// TIA Portal V21 export
FUNCTION "AlarmsFc" : Void   // FC181, LAD
{ S7_Optimized_Access := 'TRUE' }
// stored: AutoNumber false, SetENOAutomatically false
   VAR_TEMP   // added for the SCL form of the ladder/FBD networks
      _w1 : Bool;
      _w2 : Bool;
      _w3 : Bool;
      _w4 : Bool;
      _w5 : Bool;
      _w6 : Bool;
      _w7 : Bool;
      _w8 : Bool;
      _w9 : Bool;
      _w10 : Bool;
      _w11 : Bool;
      _w12 : Bool;
      _w13 : Bool;
      _w14 : Bool;
      _w15 : Bool;
      _w16 : Bool;
      _w17 : Bool;
      _w18 : Bool;
      _w19 : Bool;
      _w20 : Bool;
      _w21 : Bool;
      _w22 : Bool;
      _w23 : Bool;
      _w24 : Bool;
      _w25 : Bool;
      _w26 : Bool;
      _w27 : Bool;
      _w28 : Bool;
      _w29 : Bool;
      _w30 : Bool;
      _w31 : Bool;
      _w32 : Bool;
      _w33 : Bool;
      _w34 : Bool;
      _w35 : Bool;
      _w36 : Bool;
      _w37 : Bool;
      _w38 : Bool;
      _w39 : Bool;
      _w40 : Bool;
      _w41 : Bool;
      _w42 : Bool;
      _w43 : Bool;
      _w44 : Bool;
      _w45 : Bool;
      _w46 : Bool;
   END_VAR
BEGIN

REGION Network 1: "SafetyAlarms".ControlKeyOff
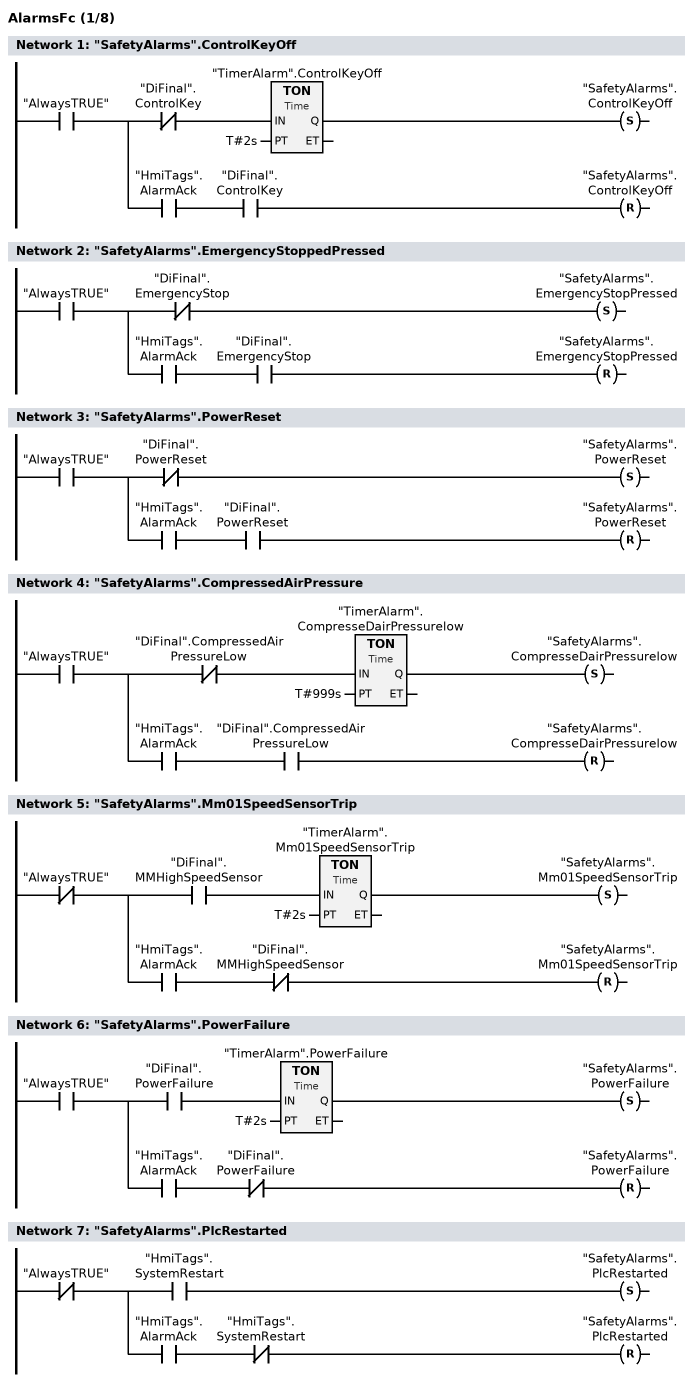
   RUNG wire#powerrail
      Contact( "AlwaysTRUE" )
      wire#w1
      I_Contact( "DiFinal".ControlKey )
      { S7_Templates := "time_type := Time" } "TimerAlarm".ControlKeyOff.TON(pt := T#2s, et =>)
      S_Coil( "SafetyAlarms".ControlKeyOff )
   END_RUNG
   RUNG wire#w1
      Contact( "HmiTags".AlarmAck )
      Contact( "DiFinal".ControlKey )
      R_Coil( "SafetyAlarms".ControlKeyOff )
   END_RUNG
   // the same network as SCL:
   "TimerAlarm".ControlKeyOff.TON(IN := "AlwaysTRUE" AND NOT "DiFinal".ControlKey, PT := T#2s);
   IF "TimerAlarm".ControlKeyOff.Q THEN "SafetyAlarms".ControlKeyOff := TRUE; END_IF;
   IF "AlwaysTRUE" AND "HmiTags".AlarmAck AND "DiFinal".ControlKey THEN
       "SafetyAlarms".ControlKeyOff := FALSE;
   END_IF;
END_REGION

REGION Network 2: "SafetyAlarms".EmergencyStoppedPressed
   RUNG wire#powerrail
      Contact( "AlwaysTRUE" )
      wire#w1
      I_Contact( "DiFinal".EmergencyStop )
      S_Coil( "SafetyAlarms".EmergencyStopPressed )
   END_RUNG
   RUNG wire#w1
      Contact( "HmiTags".AlarmAck )
      Contact( "DiFinal".EmergencyStop )
      R_Coil( "SafetyAlarms".EmergencyStopPressed )
   END_RUNG
   // the same network as SCL:
   IF "AlwaysTRUE" AND NOT "DiFinal".EmergencyStop THEN "SafetyAlarms".EmergencyStopPressed := TRUE; END_IF;
   IF "AlwaysTRUE" AND "HmiTags".AlarmAck AND "DiFinal".EmergencyStop THEN
       "SafetyAlarms".EmergencyStopPressed := FALSE;
   END_IF;
END_REGION

REGION Network 3: "SafetyAlarms".PowerReset
   RUNG wire#powerrail
      Contact( "AlwaysTRUE" )
      wire#w1
      I_Contact( "DiFinal".PowerReset )
      S_Coil( "SafetyAlarms".PowerReset )
   END_RUNG
   RUNG wire#w1
      Contact( "HmiTags".AlarmAck )
      Contact( "DiFinal".PowerReset )
      R_Coil( "SafetyAlarms".PowerReset )
   END_RUNG
   // the same network as SCL:
   IF "AlwaysTRUE" AND NOT "DiFinal".PowerReset THEN "SafetyAlarms".PowerReset := TRUE; END_IF;
   IF "AlwaysTRUE" AND "HmiTags".AlarmAck AND "DiFinal".PowerReset THEN
       "SafetyAlarms".PowerReset := FALSE;
   END_IF;
END_REGION

REGION Network 4: "SafetyAlarms".CompressedAirPressure
   RUNG wire#powerrail
      Contact( "AlwaysTRUE" )
      wire#w1
      I_Contact( "DiFinal".CompressedAirPressureLow )
      { S7_Templates := "time_type := Time" } "TimerAlarm".CompresseDairPressurelow.TON(pt := T#999s, et =>)
      S_Coil( "SafetyAlarms".CompresseDairPressurelow )
   END_RUNG
   RUNG wire#w1
      Contact( "HmiTags".AlarmAck )
      Contact( "DiFinal".CompressedAirPressureLow )
      R_Coil( "SafetyAlarms".CompresseDairPressurelow )
   END_RUNG
   // the same network as SCL:
   "TimerAlarm".CompresseDairPressurelow.TON(IN := "AlwaysTRUE" AND NOT "DiFinal".CompressedAirPressureLow,
                           PT := T#999s);
   IF "TimerAlarm".CompresseDairPressurelow.Q THEN "SafetyAlarms".CompresseDairPressurelow := TRUE; END_IF;
   IF "AlwaysTRUE" AND "HmiTags".AlarmAck AND "DiFinal".CompressedAirPressureLow THEN
       "SafetyAlarms".CompresseDairPressurelow := FALSE;
   END_IF;
END_REGION

REGION Network 5: "SafetyAlarms".Mm01SpeedSensorTrip
   RUNG wire#powerrail
      I_Contact( "AlwaysTRUE" )
      wire#w1
      Contact( "DiFinal".MMHighSpeedSensor )
      { S7_Templates := "time_type := Time" } "TimerAlarm".Mm01SpeedSensorTrip.TON(pt := T#2s, et =>)
      S_Coil( "SafetyAlarms".Mm01SpeedSensorTrip )
   END_RUNG
   RUNG wire#w1
      Contact( "HmiTags".AlarmAck )
      I_Contact( "DiFinal".MMHighSpeedSensor )
      R_Coil( "SafetyAlarms".Mm01SpeedSensorTrip )
   END_RUNG
   // the same network as SCL:
   "TimerAlarm".Mm01SpeedSensorTrip.TON(IN := NOT "AlwaysTRUE" AND "DiFinal".MMHighSpeedSensor, PT := T#2s);
   IF "TimerAlarm".Mm01SpeedSensorTrip.Q THEN "SafetyAlarms".Mm01SpeedSensorTrip := TRUE; END_IF;
   IF NOT "AlwaysTRUE" AND "HmiTags".AlarmAck AND NOT "DiFinal".MMHighSpeedSensor THEN
       "SafetyAlarms".Mm01SpeedSensorTrip := FALSE;
   END_IF;
END_REGION

REGION Network 6: "SafetyAlarms".PowerFailure
   RUNG wire#powerrail
      Contact( "AlwaysTRUE" )
      wire#w1
      Contact( "DiFinal".PowerFailure )
      { S7_Templates := "time_type := Time" } "TimerAlarm".PowerFailure.TON(pt := T#2s, et =>)
      S_Coil( "SafetyAlarms".PowerFailure )
   END_RUNG
   RUNG wire#w1
      Contact( "HmiTags".AlarmAck )
      I_Contact( "DiFinal".PowerFailure )
      R_Coil( "SafetyAlarms".PowerFailure )
   END_RUNG
   // the same network as SCL:
   "TimerAlarm".PowerFailure.TON(IN := "AlwaysTRUE" AND "DiFinal".PowerFailure, PT := T#2s);
   IF "TimerAlarm".PowerFailure.Q THEN "SafetyAlarms".PowerFailure := TRUE; END_IF;
   IF "AlwaysTRUE" AND "HmiTags".AlarmAck AND NOT "DiFinal".PowerFailure THEN
       "SafetyAlarms".PowerFailure := FALSE;
   END_IF;
END_REGION

REGION Network 7: "SafetyAlarms".PlcRestarted
   RUNG wire#powerrail
      I_Contact( "AlwaysTRUE" )
      wire#w1
      Contact( "HmiTags".SystemRestart )
      S_Coil( "SafetyAlarms".PlcRestarted )
   END_RUNG
   RUNG wire#w1
      Contact( "HmiTags".AlarmAck )
      I_Contact( "HmiTags".SystemRestart )
      R_Coil( "SafetyAlarms".PlcRestarted )
   END_RUNG
   // the same network as SCL:
   IF NOT "AlwaysTRUE" AND "HmiTags".SystemRestart THEN "SafetyAlarms".PlcRestarted := TRUE; END_IF;
   IF NOT "AlwaysTRUE" AND "HmiTags".AlarmAck AND NOT "HmiTags".SystemRestart THEN
       "SafetyAlarms".PlcRestarted := FALSE;
   END_IF;
END_REGION

REGION Network 8: "SafetyAlarms".Mm01OverloadTrip
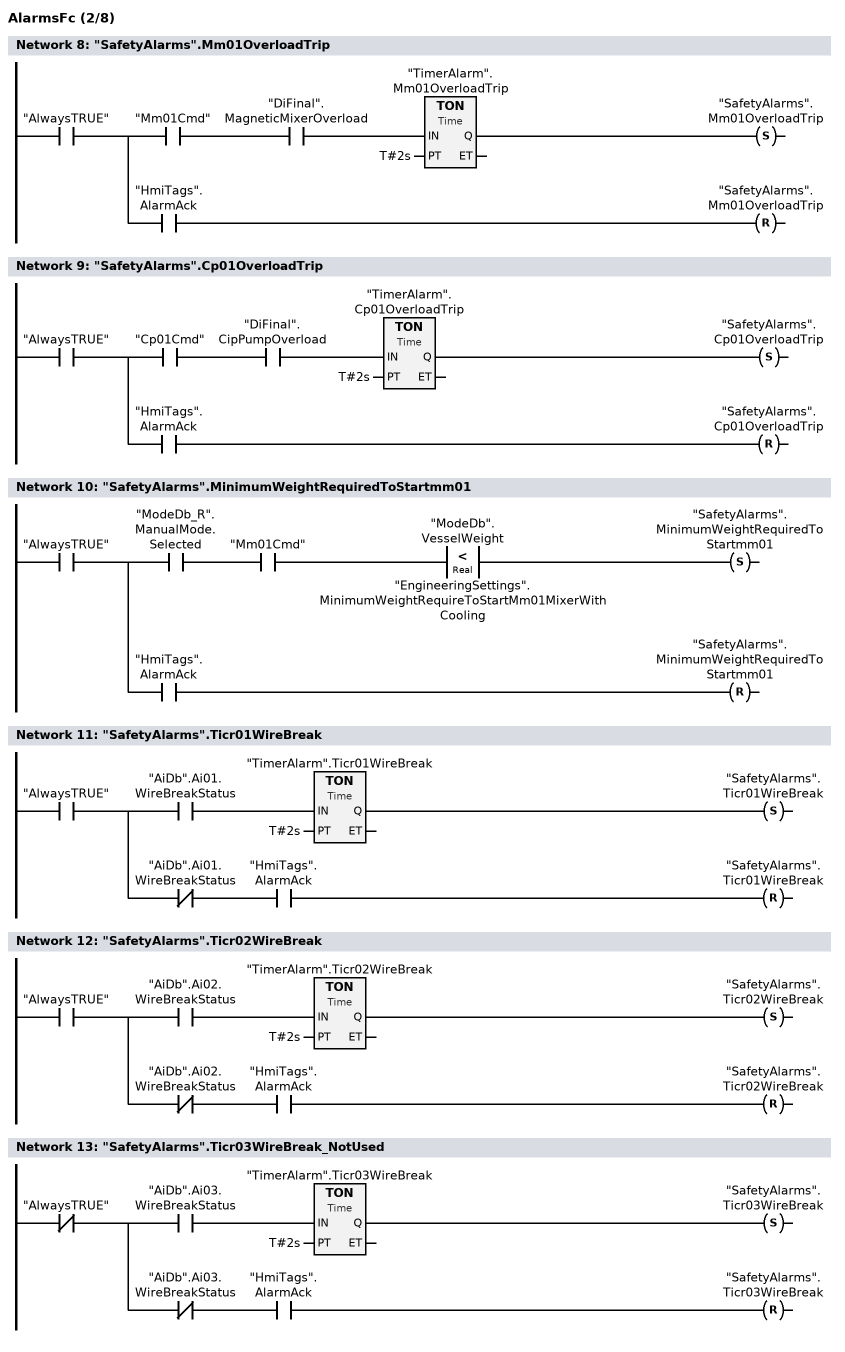
   RUNG wire#powerrail
      Contact( "AlwaysTRUE" )
      wire#w1
      Contact( "Mm01Cmd" )
      Contact( "DiFinal".MagneticMixerOverload )
      { S7_Templates := "time_type := Time" } "TimerAlarm".Mm01OverloadTrip.TON(pt := T#2s, et =>)
      S_Coil( "SafetyAlarms".Mm01OverloadTrip )
   END_RUNG
   RUNG wire#w1
      Contact( "HmiTags".AlarmAck )
      R_Coil( "SafetyAlarms".Mm01OverloadTrip )
   END_RUNG
   // the same network as SCL:
   "TimerAlarm".Mm01OverloadTrip.TON(IN := "AlwaysTRUE" AND "Mm01Cmd" AND "DiFinal".MagneticMixerOverload,
                           PT := T#2s);
   IF "TimerAlarm".Mm01OverloadTrip.Q THEN "SafetyAlarms".Mm01OverloadTrip := TRUE; END_IF;
   IF "AlwaysTRUE" AND "HmiTags".AlarmAck THEN "SafetyAlarms".Mm01OverloadTrip := FALSE; END_IF;
END_REGION

REGION Network 9: "SafetyAlarms".Cp01OverloadTrip
   RUNG wire#powerrail
      Contact( "AlwaysTRUE" )
      wire#w1
      Contact( "Cp01Cmd" )
      Contact( "DiFinal".CipPumpOverload )
      { S7_Templates := "time_type := Time" } "TimerAlarm".Cp01OverloadTrip.TON(pt := T#2s, et =>)
      S_Coil( "SafetyAlarms".Cp01OverloadTrip )
   END_RUNG
   RUNG wire#w1
      Contact( "HmiTags".AlarmAck )
      R_Coil( "SafetyAlarms".Cp01OverloadTrip )
   END_RUNG
   // the same network as SCL:
   "TimerAlarm".Cp01OverloadTrip.TON(IN := "AlwaysTRUE" AND "Cp01Cmd" AND "DiFinal".CipPumpOverload, PT := T#2s);
   IF "TimerAlarm".Cp01OverloadTrip.Q THEN "SafetyAlarms".Cp01OverloadTrip := TRUE; END_IF;
   IF "AlwaysTRUE" AND "HmiTags".AlarmAck THEN "SafetyAlarms".Cp01OverloadTrip := FALSE; END_IF;
END_REGION

REGION Network 10: "SafetyAlarms".MinimumWeightRequiredToStartmm01
   RUNG wire#powerrail
      Contact( "AlwaysTRUE" )
      wire#w1
      Contact( "ModeDb_R".ManualMode.Selected )
      Contact( "Mm01Cmd" )
      { S7_Templates := "SrcType := Real" } LT_Contact(in1 := "ModeDb".VesselWeight, in2 := "EngineeringSettings".MinimumWeightRequireToStartMm01MixerWithCooling)
      S_Coil( "SafetyAlarms".MinimumWeightRequiredToStartmm01 )
   END_RUNG
   RUNG wire#w1
      Contact( "HmiTags".AlarmAck )
      R_Coil( "SafetyAlarms".MinimumWeightRequiredToStartmm01 )
   END_RUNG
   // the same network as SCL:
   IF "AlwaysTRUE" AND "ModeDb_R".ManualMode.Selected AND "Mm01Cmd" AND ("ModeDb".VesselWeight < "EngineeringSettings".MinimumWeightRequireToStartMm01MixerWithCooling) THEN
       "SafetyAlarms".MinimumWeightRequiredToStartmm01 := TRUE;
   END_IF;
   IF "AlwaysTRUE" AND "HmiTags".AlarmAck THEN
       "SafetyAlarms".MinimumWeightRequiredToStartmm01 := FALSE;
   END_IF;
END_REGION

REGION Network 11: "SafetyAlarms".Ticr01WireBreak
   RUNG wire#powerrail
      Contact( "AlwaysTRUE" )
      wire#w1
      Contact( "AiDb".Ai01.WireBreakStatus )
      { S7_Templates := "time_type := Time" } "TimerAlarm".Ticr01WireBreak.TON(pt := T#2s, et =>)
      S_Coil( "SafetyAlarms".Ticr01WireBreak )
   END_RUNG
   RUNG wire#w1
      I_Contact( "AiDb".Ai01.WireBreakStatus )
      Contact( "HmiTags".AlarmAck )
      R_Coil( "SafetyAlarms".Ticr01WireBreak )
   END_RUNG
   // the same network as SCL:
   "TimerAlarm".Ticr01WireBreak.TON(IN := "AlwaysTRUE" AND "AiDb".Ai01.WireBreakStatus, PT := T#2s);
   IF "TimerAlarm".Ticr01WireBreak.Q THEN "SafetyAlarms".Ticr01WireBreak := TRUE; END_IF;
   IF "AlwaysTRUE" AND NOT "AiDb".Ai01.WireBreakStatus AND "HmiTags".AlarmAck THEN
       "SafetyAlarms".Ticr01WireBreak := FALSE;
   END_IF;
END_REGION

REGION Network 12: "SafetyAlarms".Ticr02WireBreak
   RUNG wire#powerrail
      Contact( "AlwaysTRUE" )
      wire#w1
      Contact( "AiDb".Ai02.WireBreakStatus )
      { S7_Templates := "time_type := Time" } "TimerAlarm".Ticr02WireBreak.TON(pt := T#2s, et =>)
      S_Coil( "SafetyAlarms".Ticr02WireBreak )
   END_RUNG
   RUNG wire#w1
      I_Contact( "AiDb".Ai02.WireBreakStatus )
      Contact( "HmiTags".AlarmAck )
      R_Coil( "SafetyAlarms".Ticr02WireBreak )
   END_RUNG
   // the same network as SCL:
   "TimerAlarm".Ticr02WireBreak.TON(IN := "AlwaysTRUE" AND "AiDb".Ai02.WireBreakStatus, PT := T#2s);
   IF "TimerAlarm".Ticr02WireBreak.Q THEN "SafetyAlarms".Ticr02WireBreak := TRUE; END_IF;
   IF "AlwaysTRUE" AND NOT "AiDb".Ai02.WireBreakStatus AND "HmiTags".AlarmAck THEN
       "SafetyAlarms".Ticr02WireBreak := FALSE;
   END_IF;
END_REGION

REGION Network 13: "SafetyAlarms".Ticr03WireBreak_NotUsed
   RUNG wire#powerrail
      I_Contact( "AlwaysTRUE" )
      wire#w1
      Contact( "AiDb".Ai03.WireBreakStatus )
      { S7_Templates := "time_type := Time" } "TimerAlarm".Ticr03WireBreak.TON(pt := T#2s, et =>)
      S_Coil( "SafetyAlarms".Ticr03WireBreak )
   END_RUNG
   RUNG wire#w1
      I_Contact( "AiDb".Ai03.WireBreakStatus )
      Contact( "HmiTags".AlarmAck )
      R_Coil( "SafetyAlarms".Ticr03WireBreak )
   END_RUNG
   // the same network as SCL:
   "TimerAlarm".Ticr03WireBreak.TON(IN := NOT "AlwaysTRUE" AND "AiDb".Ai03.WireBreakStatus, PT := T#2s);
   IF "TimerAlarm".Ticr03WireBreak.Q THEN "SafetyAlarms".Ticr03WireBreak := TRUE; END_IF;
   IF NOT "AlwaysTRUE" AND NOT "AiDb".Ai03.WireBreakStatus AND "HmiTags".AlarmAck THEN
       "SafetyAlarms".Ticr03WireBreak := FALSE;
   END_IF;
END_REGION

REGION Network 14: "SafetyAlarms".Ticr04WireBreak_NotUsed
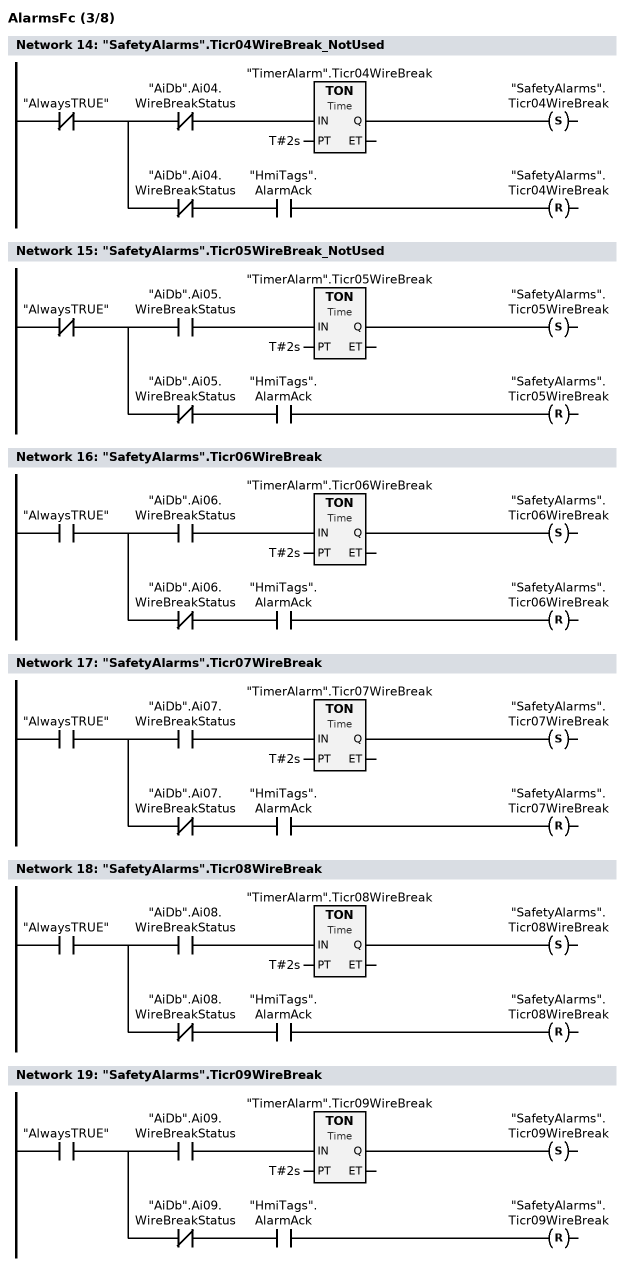
   RUNG wire#powerrail
      I_Contact( "AlwaysTRUE" )
      wire#w1
      I_Contact( "AiDb".Ai04.WireBreakStatus )
      { S7_Templates := "time_type := Time" } "TimerAlarm".Ticr04WireBreak.TON(pt := T#2s, et =>)
      S_Coil( "SafetyAlarms".Ticr04WireBreak )
   END_RUNG
   RUNG wire#w1
      I_Contact( "AiDb".Ai04.WireBreakStatus )
      Contact( "HmiTags".AlarmAck )
      R_Coil( "SafetyAlarms".Ticr04WireBreak )
   END_RUNG
   // the same network as SCL:
   "TimerAlarm".Ticr04WireBreak.TON(IN := NOT "AlwaysTRUE" AND NOT "AiDb".Ai04.WireBreakStatus, PT := T#2s);
   IF "TimerAlarm".Ticr04WireBreak.Q THEN "SafetyAlarms".Ticr04WireBreak := TRUE; END_IF;
   IF NOT "AlwaysTRUE" AND NOT "AiDb".Ai04.WireBreakStatus AND "HmiTags".AlarmAck THEN
       "SafetyAlarms".Ticr04WireBreak := FALSE;
   END_IF;
END_REGION

REGION Network 15: "SafetyAlarms".Ticr05WireBreak_NotUsed
   RUNG wire#powerrail
      I_Contact( "AlwaysTRUE" )
      wire#w1
      Contact( "AiDb".Ai05.WireBreakStatus )
      { S7_Templates := "time_type := Time" } "TimerAlarm".Ticr05WireBreak.TON(pt := T#2s, et =>)
      S_Coil( "SafetyAlarms".Ticr05WireBreak )
   END_RUNG
   RUNG wire#w1
      I_Contact( "AiDb".Ai05.WireBreakStatus )
      Contact( "HmiTags".AlarmAck )
      R_Coil( "SafetyAlarms".Ticr05WireBreak )
   END_RUNG
   // the same network as SCL:
   "TimerAlarm".Ticr05WireBreak.TON(IN := NOT "AlwaysTRUE" AND "AiDb".Ai05.WireBreakStatus, PT := T#2s);
   IF "TimerAlarm".Ticr05WireBreak.Q THEN "SafetyAlarms".Ticr05WireBreak := TRUE; END_IF;
   IF NOT "AlwaysTRUE" AND NOT "AiDb".Ai05.WireBreakStatus AND "HmiTags".AlarmAck THEN
       "SafetyAlarms".Ticr05WireBreak := FALSE;
   END_IF;
END_REGION

REGION Network 16: "SafetyAlarms".Ticr06WireBreak
   RUNG wire#powerrail
      Contact( "AlwaysTRUE" )
      wire#w1
      Contact( "AiDb".Ai06.WireBreakStatus )
      { S7_Templates := "time_type := Time" } "TimerAlarm".Ticr06WireBreak.TON(pt := T#2s, et =>)
      S_Coil( "SafetyAlarms".Ticr06WireBreak )
   END_RUNG
   RUNG wire#w1
      I_Contact( "AiDb".Ai06.WireBreakStatus )
      Contact( "HmiTags".AlarmAck )
      R_Coil( "SafetyAlarms".Ticr06WireBreak )
   END_RUNG
   // the same network as SCL:
   "TimerAlarm".Ticr06WireBreak.TON(IN := "AlwaysTRUE" AND "AiDb".Ai06.WireBreakStatus, PT := T#2s);
   IF "TimerAlarm".Ticr06WireBreak.Q THEN "SafetyAlarms".Ticr06WireBreak := TRUE; END_IF;
   IF "AlwaysTRUE" AND NOT "AiDb".Ai06.WireBreakStatus AND "HmiTags".AlarmAck THEN
       "SafetyAlarms".Ticr06WireBreak := FALSE;
   END_IF;
END_REGION

REGION Network 17: "SafetyAlarms".Ticr07WireBreak
   RUNG wire#powerrail
      Contact( "AlwaysTRUE" )
      wire#w1
      Contact( "AiDb".Ai07.WireBreakStatus )
      { S7_Templates := "time_type := Time" } "TimerAlarm".Ticr07WireBreak.TON(pt := T#2s, et =>)
      S_Coil( "SafetyAlarms".Ticr07WireBreak )
   END_RUNG
   RUNG wire#w1
      I_Contact( "AiDb".Ai07.WireBreakStatus )
      Contact( "HmiTags".AlarmAck )
      R_Coil( "SafetyAlarms".Ticr07WireBreak )
   END_RUNG
   // the same network as SCL:
   "TimerAlarm".Ticr07WireBreak.TON(IN := "AlwaysTRUE" AND "AiDb".Ai07.WireBreakStatus, PT := T#2s);
   IF "TimerAlarm".Ticr07WireBreak.Q THEN "SafetyAlarms".Ticr07WireBreak := TRUE; END_IF;
   IF "AlwaysTRUE" AND NOT "AiDb".Ai07.WireBreakStatus AND "HmiTags".AlarmAck THEN
       "SafetyAlarms".Ticr07WireBreak := FALSE;
   END_IF;
END_REGION

REGION Network 18: "SafetyAlarms".Ticr08WireBreak
   RUNG wire#powerrail
      Contact( "AlwaysTRUE" )
      wire#w1
      Contact( "AiDb".Ai08.WireBreakStatus )
      { S7_Templates := "time_type := Time" } "TimerAlarm".Ticr08WireBreak.TON(pt := T#2s, et =>)
      S_Coil( "SafetyAlarms".Ticr08WireBreak )
   END_RUNG
   RUNG wire#w1
      I_Contact( "AiDb".Ai08.WireBreakStatus )
      Contact( "HmiTags".AlarmAck )
      R_Coil( "SafetyAlarms".Ticr08WireBreak )
   END_RUNG
   // the same network as SCL:
   "TimerAlarm".Ticr08WireBreak.TON(IN := "AlwaysTRUE" AND "AiDb".Ai08.WireBreakStatus, PT := T#2s);
   IF "TimerAlarm".Ticr08WireBreak.Q THEN "SafetyAlarms".Ticr08WireBreak := TRUE; END_IF;
   IF "AlwaysTRUE" AND NOT "AiDb".Ai08.WireBreakStatus AND "HmiTags".AlarmAck THEN
       "SafetyAlarms".Ticr08WireBreak := FALSE;
   END_IF;
END_REGION

REGION Network 19: "SafetyAlarms".Ticr09WireBreak
   RUNG wire#powerrail
      Contact( "AlwaysTRUE" )
      wire#w1
      Contact( "AiDb".Ai09.WireBreakStatus )
      { S7_Templates := "time_type := Time" } "TimerAlarm".Ticr09WireBreak.TON(pt := T#2s, et =>)
      S_Coil( "SafetyAlarms".Ticr09WireBreak )
   END_RUNG
   RUNG wire#w1
      I_Contact( "AiDb".Ai09.WireBreakStatus )
      Contact( "HmiTags".AlarmAck )
      R_Coil( "SafetyAlarms".Ticr09WireBreak )
   END_RUNG
   // the same network as SCL:
   "TimerAlarm".Ticr09WireBreak.TON(IN := "AlwaysTRUE" AND "AiDb".Ai09.WireBreakStatus, PT := T#2s);
   IF "TimerAlarm".Ticr09WireBreak.Q THEN "SafetyAlarms".Ticr09WireBreak := TRUE; END_IF;
   IF "AlwaysTRUE" AND NOT "AiDb".Ai09.WireBreakStatus AND "HmiTags".AlarmAck THEN
       "SafetyAlarms".Ticr09WireBreak := FALSE;
   END_IF;
END_REGION

REGION Network 20: "SafetyAlarms".Ticr10WireBreak
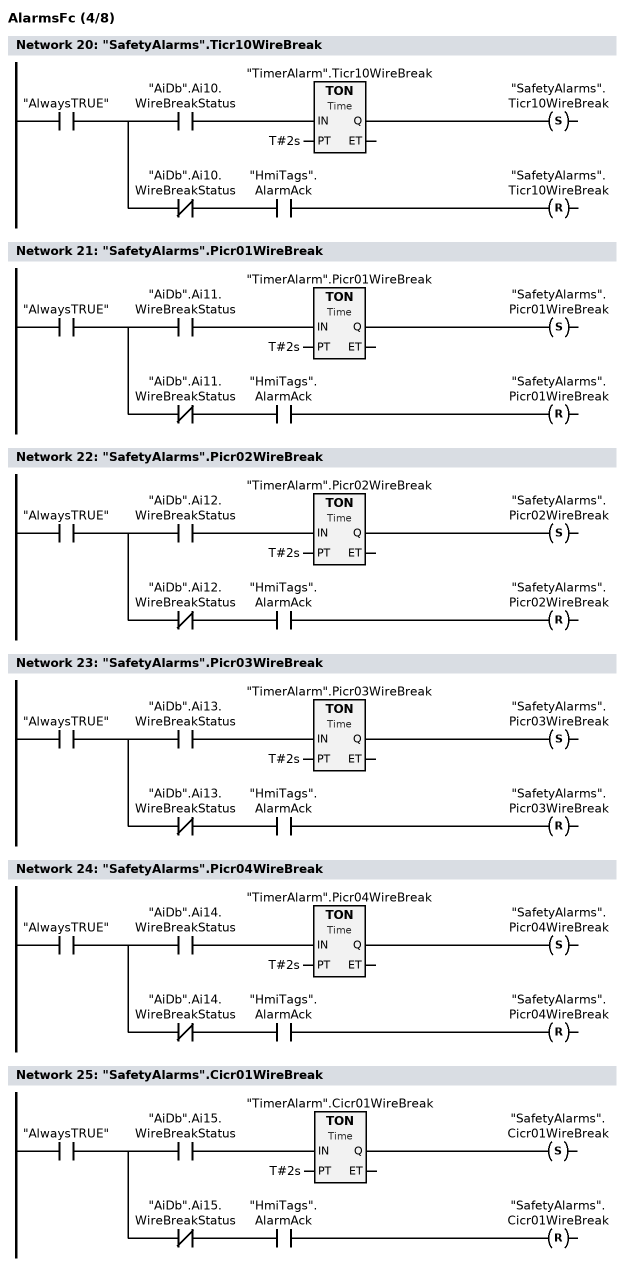
   RUNG wire#powerrail
      Contact( "AlwaysTRUE" )
      wire#w1
      Contact( "AiDb".Ai10.WireBreakStatus )
      { S7_Templates := "time_type := Time" } "TimerAlarm".Ticr10WireBreak.TON(pt := T#2s, et =>)
      S_Coil( "SafetyAlarms".Ticr10WireBreak )
   END_RUNG
   RUNG wire#w1
      I_Contact( "AiDb".Ai10.WireBreakStatus )
      Contact( "HmiTags".AlarmAck )
      R_Coil( "SafetyAlarms".Ticr10WireBreak )
   END_RUNG
   // the same network as SCL:
   "TimerAlarm".Ticr10WireBreak.TON(IN := "AlwaysTRUE" AND "AiDb".Ai10.WireBreakStatus, PT := T#2s);
   IF "TimerAlarm".Ticr10WireBreak.Q THEN "SafetyAlarms".Ticr10WireBreak := TRUE; END_IF;
   IF "AlwaysTRUE" AND NOT "AiDb".Ai10.WireBreakStatus AND "HmiTags".AlarmAck THEN
       "SafetyAlarms".Ticr10WireBreak := FALSE;
   END_IF;
END_REGION

REGION Network 21: "SafetyAlarms".Picr01WireBreak
   RUNG wire#powerrail
      Contact( "AlwaysTRUE" )
      wire#w1
      Contact( "AiDb".Ai11.WireBreakStatus )
      { S7_Templates := "time_type := Time" } "TimerAlarm".Picr01WireBreak.TON(pt := T#2s, et =>)
      S_Coil( "SafetyAlarms".Picr01WireBreak )
   END_RUNG
   RUNG wire#w1
      I_Contact( "AiDb".Ai11.WireBreakStatus )
      Contact( "HmiTags".AlarmAck )
      R_Coil( "SafetyAlarms".Picr01WireBreak )
   END_RUNG
   // the same network as SCL:
   "TimerAlarm".Picr01WireBreak.TON(IN := "AlwaysTRUE" AND "AiDb".Ai11.WireBreakStatus, PT := T#2s);
   IF "TimerAlarm".Picr01WireBreak.Q THEN "SafetyAlarms".Picr01WireBreak := TRUE; END_IF;
   IF "AlwaysTRUE" AND NOT "AiDb".Ai11.WireBreakStatus AND "HmiTags".AlarmAck THEN
       "SafetyAlarms".Picr01WireBreak := FALSE;
   END_IF;
END_REGION

REGION Network 22: "SafetyAlarms".Picr02WireBreak
   RUNG wire#powerrail
      Contact( "AlwaysTRUE" )
      wire#w1
      Contact( "AiDb".Ai12.WireBreakStatus )
      { S7_Templates := "time_type := Time" } "TimerAlarm".Picr02WireBreak.TON(pt := T#2s, et =>)
      S_Coil( "SafetyAlarms".Picr02WireBreak )
   END_RUNG
   RUNG wire#w1
      I_Contact( "AiDb".Ai12.WireBreakStatus )
      Contact( "HmiTags".AlarmAck )
      R_Coil( "SafetyAlarms".Picr02WireBreak )
   END_RUNG
   // the same network as SCL:
   "TimerAlarm".Picr02WireBreak.TON(IN := "AlwaysTRUE" AND "AiDb".Ai12.WireBreakStatus, PT := T#2s);
   IF "TimerAlarm".Picr02WireBreak.Q THEN "SafetyAlarms".Picr02WireBreak := TRUE; END_IF;
   IF "AlwaysTRUE" AND NOT "AiDb".Ai12.WireBreakStatus AND "HmiTags".AlarmAck THEN
       "SafetyAlarms".Picr02WireBreak := FALSE;
   END_IF;
END_REGION

REGION Network 23: "SafetyAlarms".Picr03WireBreak
   RUNG wire#powerrail
      Contact( "AlwaysTRUE" )
      wire#w1
      Contact( "AiDb".Ai13.WireBreakStatus )
      { S7_Templates := "time_type := Time" } "TimerAlarm".Picr03WireBreak.TON(pt := T#2s, et =>)
      S_Coil( "SafetyAlarms".Picr03WireBreak )
   END_RUNG
   RUNG wire#w1
      I_Contact( "AiDb".Ai13.WireBreakStatus )
      Contact( "HmiTags".AlarmAck )
      R_Coil( "SafetyAlarms".Picr03WireBreak )
   END_RUNG
   // the same network as SCL:
   "TimerAlarm".Picr03WireBreak.TON(IN := "AlwaysTRUE" AND "AiDb".Ai13.WireBreakStatus, PT := T#2s);
   IF "TimerAlarm".Picr03WireBreak.Q THEN "SafetyAlarms".Picr03WireBreak := TRUE; END_IF;
   IF "AlwaysTRUE" AND NOT "AiDb".Ai13.WireBreakStatus AND "HmiTags".AlarmAck THEN
       "SafetyAlarms".Picr03WireBreak := FALSE;
   END_IF;
END_REGION

REGION Network 24: "SafetyAlarms".Picr04WireBreak
   RUNG wire#powerrail
      Contact( "AlwaysTRUE" )
      wire#w1
      Contact( "AiDb".Ai14.WireBreakStatus )
      { S7_Templates := "time_type := Time" } "TimerAlarm".Picr04WireBreak.TON(pt := T#2s, et =>)
      S_Coil( "SafetyAlarms".Picr04WireBreak )
   END_RUNG
   RUNG wire#w1
      I_Contact( "AiDb".Ai14.WireBreakStatus )
      Contact( "HmiTags".AlarmAck )
      R_Coil( "SafetyAlarms".Picr04WireBreak )
   END_RUNG
   // the same network as SCL:
   "TimerAlarm".Picr04WireBreak.TON(IN := "AlwaysTRUE" AND "AiDb".Ai14.WireBreakStatus, PT := T#2s);
   IF "TimerAlarm".Picr04WireBreak.Q THEN "SafetyAlarms".Picr04WireBreak := TRUE; END_IF;
   IF "AlwaysTRUE" AND NOT "AiDb".Ai14.WireBreakStatus AND "HmiTags".AlarmAck THEN
       "SafetyAlarms".Picr04WireBreak := FALSE;
   END_IF;
END_REGION

REGION Network 25: "SafetyAlarms".Cicr01WireBreak
   RUNG wire#powerrail
      Contact( "AlwaysTRUE" )
      wire#w1
      Contact( "AiDb".Ai15.WireBreakStatus )
      { S7_Templates := "time_type := Time" } "TimerAlarm".Cicr01WireBreak.TON(pt := T#2s, et =>)
      S_Coil( "SafetyAlarms".Cicr01WireBreak )
   END_RUNG
   RUNG wire#w1
      I_Contact( "AiDb".Ai15.WireBreakStatus )
      Contact( "HmiTags".AlarmAck )
      R_Coil( "SafetyAlarms".Cicr01WireBreak )
   END_RUNG
   // the same network as SCL:
   "TimerAlarm".Cicr01WireBreak.TON(IN := "AlwaysTRUE" AND "AiDb".Ai15.WireBreakStatus, PT := T#2s);
   IF "TimerAlarm".Cicr01WireBreak.Q THEN "SafetyAlarms".Cicr01WireBreak := TRUE; END_IF;
   IF "AlwaysTRUE" AND NOT "AiDb".Ai15.WireBreakStatus AND "HmiTags".AlarmAck THEN
       "SafetyAlarms".Cicr01WireBreak := FALSE;
   END_IF;
END_REGION

REGION Network 26: "SafetyAlarms".Lc01CommunicationFailed
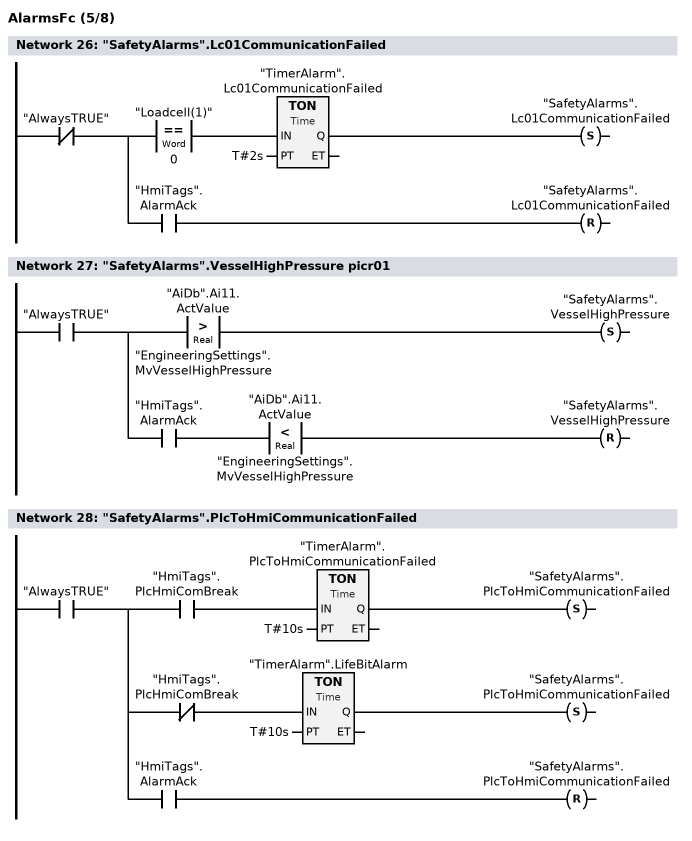
   RUNG wire#powerrail
      I_Contact( "AlwaysTRUE" )
      wire#w1
      { S7_Templates := "SrcType := Word" } EQ_Contact(in1 := "Loadcell(1)", in2 := 0)
      { S7_Templates := "time_type := Time" } "TimerAlarm".Lc01CommunicationFailed.TON(pt := T#2s, et =>)
      S_Coil( "SafetyAlarms".Lc01CommunicationFailed )
   END_RUNG
   RUNG wire#w1
      Contact( "HmiTags".AlarmAck )
      R_Coil( "SafetyAlarms".Lc01CommunicationFailed )
   END_RUNG
   // the same network as SCL:
   "TimerAlarm".Lc01CommunicationFailed.TON(IN := NOT "AlwaysTRUE" AND ("Loadcell(1)" = 0), PT := T#2s);
   IF "TimerAlarm".Lc01CommunicationFailed.Q THEN "SafetyAlarms".Lc01CommunicationFailed := TRUE; END_IF;
   IF NOT "AlwaysTRUE" AND "HmiTags".AlarmAck THEN "SafetyAlarms".Lc01CommunicationFailed := FALSE; END_IF;
END_REGION

REGION Network 27: "SafetyAlarms".VesselHighPressure picr01
   RUNG wire#powerrail
      Contact( "AlwaysTRUE" )
      wire#w1
      { S7_Templates := "SrcType := Real" } GT_Contact(in1 := "AiDb".Ai11.ActValue, in2 := "EngineeringSettings".MvVesselHighPressure)
      S_Coil( "SafetyAlarms".VesselHighPressure )
   END_RUNG
   RUNG wire#w1
      Contact( "HmiTags".AlarmAck )
      { S7_Templates := "SrcType := Real" } LT_Contact(in1 := "AiDb".Ai11.ActValue, in2 := "EngineeringSettings".MvVesselHighPressure)
      R_Coil( "SafetyAlarms".VesselHighPressure )
   END_RUNG
   // the same network as SCL:
   IF "AlwaysTRUE" AND ("AiDb".Ai11.ActValue > "EngineeringSettings".MvVesselHighPressure) THEN
       "SafetyAlarms".VesselHighPressure := TRUE;
   END_IF;
   IF "AlwaysTRUE" AND "HmiTags".AlarmAck AND ("AiDb".Ai11.ActValue < "EngineeringSettings".MvVesselHighPressure) THEN
       "SafetyAlarms".VesselHighPressure := FALSE;
   END_IF;
END_REGION

REGION Network 28: "SafetyAlarms".PlcToHmiCommunicationFailed
   RUNG wire#powerrail
      Contact( "AlwaysTRUE" )
      wire#w1
      Contact( "HmiTags".PlcHmiComBreak )
      { S7_Templates := "time_type := Time" } "TimerAlarm".PlcToHmiCommunicationFailed.TON(pt := T#10s, et =>)
      S_Coil( "SafetyAlarms".PlcToHmiCommunicationFailed )
   END_RUNG
   RUNG wire#w1
      I_Contact( "HmiTags".PlcHmiComBreak )
      { S7_Templates := "time_type := Time" } "TimerAlarm".LifeBitAlarm.TON(pt := T#10s, et =>)
      S_Coil( "SafetyAlarms".PlcToHmiCommunicationFailed )
   END_RUNG
   RUNG wire#w1
      Contact( "HmiTags".AlarmAck )
      R_Coil( "SafetyAlarms".PlcToHmiCommunicationFailed )
   END_RUNG
   // the same network as SCL:
   "TimerAlarm".PlcToHmiCommunicationFailed.TON(IN := "AlwaysTRUE" AND "HmiTags".PlcHmiComBreak, PT := T#10s);
   IF "TimerAlarm".PlcToHmiCommunicationFailed.Q THEN
       "SafetyAlarms".PlcToHmiCommunicationFailed := TRUE;
   END_IF;
   "TimerAlarm".LifeBitAlarm.TON(IN := "AlwaysTRUE" AND NOT "HmiTags".PlcHmiComBreak, PT := T#10s);
   IF "TimerAlarm".LifeBitAlarm.Q THEN "SafetyAlarms".PlcToHmiCommunicationFailed := TRUE; END_IF;
   IF "AlwaysTRUE" AND "HmiTags".AlarmAck THEN "SafetyAlarms".PlcToHmiCommunicationFailed := FALSE; END_IF;
END_REGION

REGION Network 29: "HmiTags".ManualModeFAULT
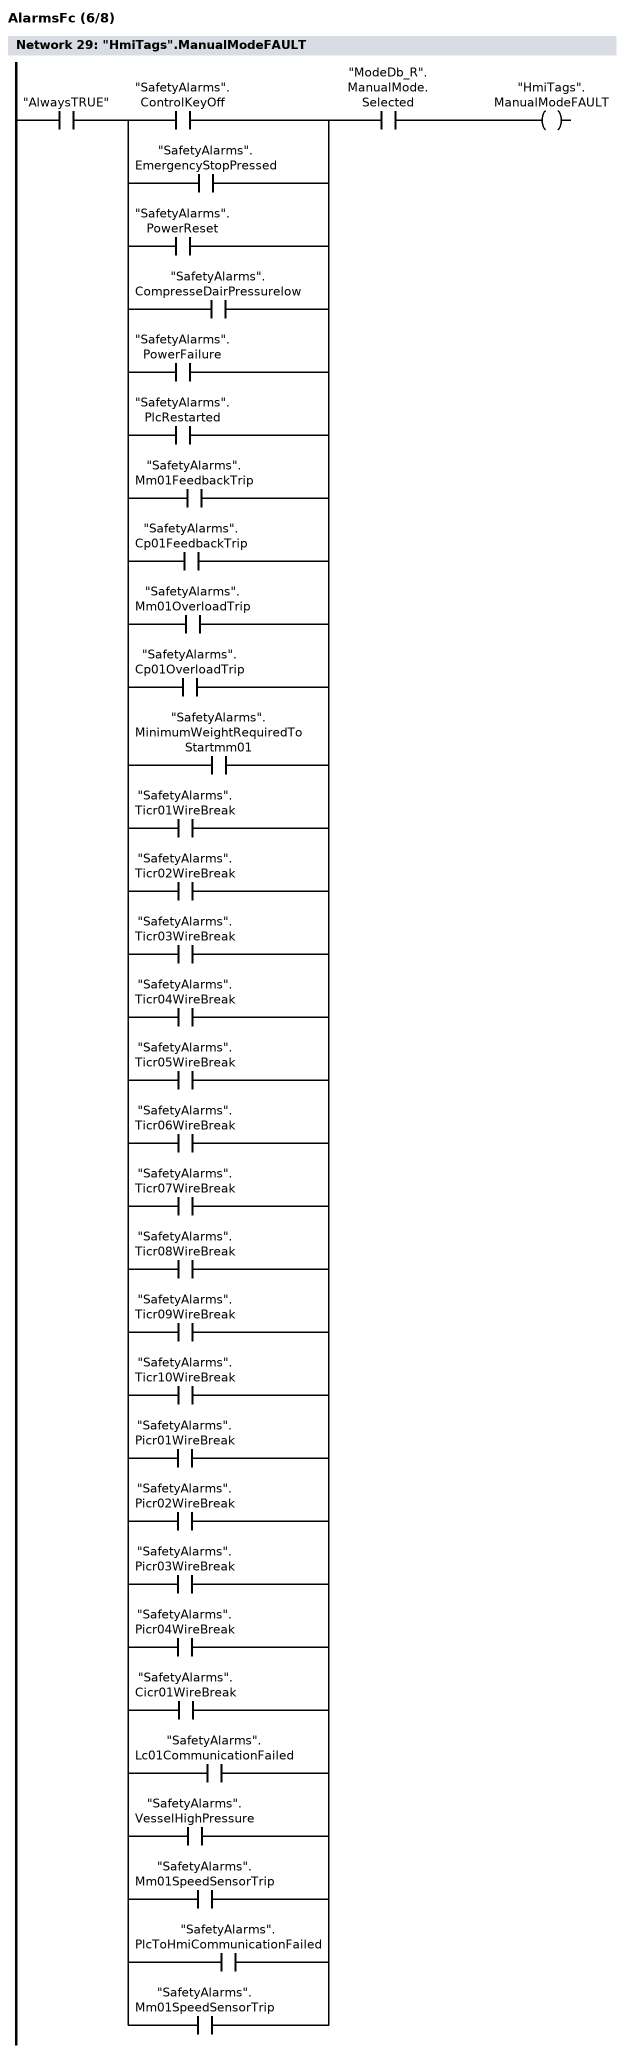
   RUNG wire#powerrail
      Contact( "AlwaysTRUE" )
      wire#w1
      Contact( "SafetyAlarms".ControlKeyOff )
      wire#w2
      Contact( "ModeDb_R".ManualMode.Selected )
      Coil( "HmiTags".ManualModeFAULT )
   END_RUNG
   RUNG wire#w1
      Contact( "SafetyAlarms".EmergencyStopPressed )
   END_RUNG wire#w2
   RUNG wire#w1
      Contact( "SafetyAlarms".PowerReset )
   END_RUNG wire#w2
   RUNG wire#w1
      Contact( "SafetyAlarms".CompresseDairPressurelow )
   END_RUNG wire#w2
   RUNG wire#w1
      Contact( "SafetyAlarms".PowerFailure )
   END_RUNG wire#w2
   RUNG wire#w1
      Contact( "SafetyAlarms".PlcRestarted )
   END_RUNG wire#w2
   RUNG wire#w1
      Contact( "SafetyAlarms".Mm01FeedbackTrip )
   END_RUNG wire#w2
   RUNG wire#w1
      Contact( "SafetyAlarms".Cp01FeedbackTrip )
   END_RUNG wire#w2
   RUNG wire#w1
      Contact( "SafetyAlarms".Mm01OverloadTrip )
   END_RUNG wire#w2
   RUNG wire#w1
      Contact( "SafetyAlarms".Cp01OverloadTrip )
   END_RUNG wire#w2
   RUNG wire#w1
      Contact( "SafetyAlarms".MinimumWeightRequiredToStartmm01 )
   END_RUNG wire#w2
   RUNG wire#w1
      Contact( "SafetyAlarms".Ticr01WireBreak )
   END_RUNG wire#w2
   RUNG wire#w1
      Contact( "SafetyAlarms".Ticr02WireBreak )
   END_RUNG wire#w2
   RUNG wire#w1
      Contact( "SafetyAlarms".Ticr03WireBreak )
   END_RUNG wire#w2
   RUNG wire#w1
      Contact( "SafetyAlarms".Ticr04WireBreak )
   END_RUNG wire#w2
   RUNG wire#w1
      Contact( "SafetyAlarms".Ticr05WireBreak )
   END_RUNG wire#w2
   RUNG wire#w1
      Contact( "SafetyAlarms".Ticr06WireBreak )
   END_RUNG wire#w2
   RUNG wire#w1
      Contact( "SafetyAlarms".Ticr07WireBreak )
   END_RUNG wire#w2
   RUNG wire#w1
      Contact( "SafetyAlarms".Ticr08WireBreak )
   END_RUNG wire#w2
   RUNG wire#w1
      Contact( "SafetyAlarms".Ticr09WireBreak )
   END_RUNG wire#w2
   RUNG wire#w1
      Contact( "SafetyAlarms".Ticr10WireBreak )
   END_RUNG wire#w2
   RUNG wire#w1
      Contact( "SafetyAlarms".Picr01WireBreak )
   END_RUNG wire#w2
   RUNG wire#w1
      Contact( "SafetyAlarms".Picr02WireBreak )
   END_RUNG wire#w2
   RUNG wire#w1
      Contact( "SafetyAlarms".Picr03WireBreak )
   END_RUNG wire#w2
   RUNG wire#w1
      Contact( "SafetyAlarms".Picr04WireBreak )
   END_RUNG wire#w2
   RUNG wire#w1
      Contact( "SafetyAlarms".Cicr01WireBreak )
   END_RUNG wire#w2
   RUNG wire#w1
      Contact( "SafetyAlarms".Lc01CommunicationFailed )
   END_RUNG wire#w2
   RUNG wire#w1
      Contact( "SafetyAlarms".VesselHighPressure )
   END_RUNG wire#w2
   RUNG wire#w1
      Contact( "SafetyAlarms".Mm01SpeedSensorTrip )
   END_RUNG wire#w2
   RUNG wire#w1
      Contact( "SafetyAlarms".PlcToHmiCommunicationFailed )
   END_RUNG wire#w2
   RUNG wire#w1
      Contact( "SafetyAlarms".Mm01SpeedSensorTrip )
   END_RUNG wire#w2
   // the same network as SCL:
   "HmiTags".ManualModeFAULT := "AlwaysTRUE" AND ("SafetyAlarms".ControlKeyOff OR "SafetyAlarms".EmergencyStopPressed OR "SafetyAlarms".PowerReset OR "SafetyAlarms".CompresseDairPressurelow OR "SafetyAlarms".PowerFailure OR "SafetyAlarms".PlcRestarted OR "SafetyAlarms".Mm01FeedbackTrip OR "SafetyAlarms".Cp01FeedbackTrip OR "SafetyAlarms".Mm01OverloadTrip OR "SafetyAlarms".Cp01OverloadTrip OR "SafetyAlarms".MinimumWeightRequiredToStartmm01 OR "SafetyAlarms".Ticr01WireBreak OR "SafetyAlarms".Ticr02WireBreak OR "SafetyAlarms".Ticr03WireBreak OR "SafetyAlarms".Ticr04WireBreak OR "SafetyAlarms".Ticr05WireBreak OR "SafetyAlarms".Ticr06WireBreak OR "SafetyAlarms".Ticr07WireBreak OR "SafetyAlarms".Ticr08WireBreak OR "SafetyAlarms".Ticr09WireBreak OR "SafetyAlarms".Ticr10WireBreak OR "SafetyAlarms".Picr01WireBreak OR "SafetyAlarms".Picr02WireBreak OR "SafetyAlarms".Picr03WireBreak OR "SafetyAlarms".Picr04WireBreak OR "SafetyAlarms".Cicr01WireBreak OR "SafetyAlarms".Lc01CommunicationFailed OR "SafetyAlarms".VesselHighPressure OR "SafetyAlarms".Mm01SpeedSensorTrip OR "SafetyAlarms".PlcToHmiCommunicationFailed OR "SafetyAlarms".Mm01SpeedSensorTrip) AND "ModeDb_R".ManualMode.Selected;
END_REGION

REGION Network 30: "HmiTags".Hooter -- set
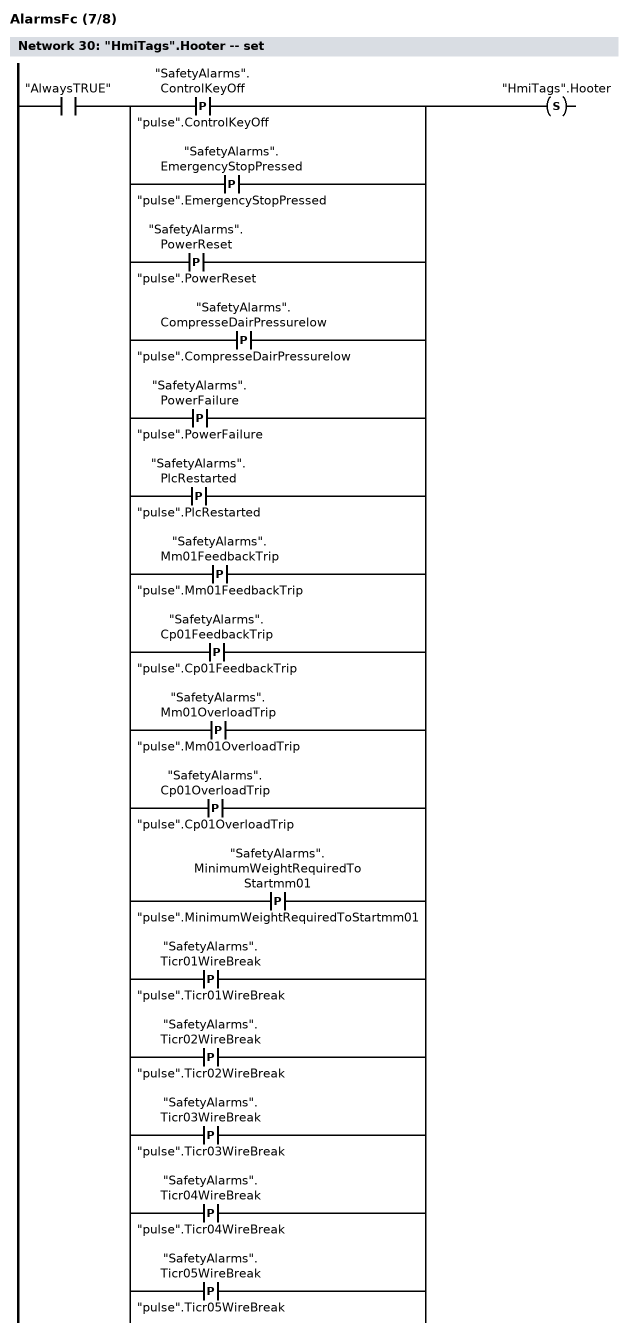
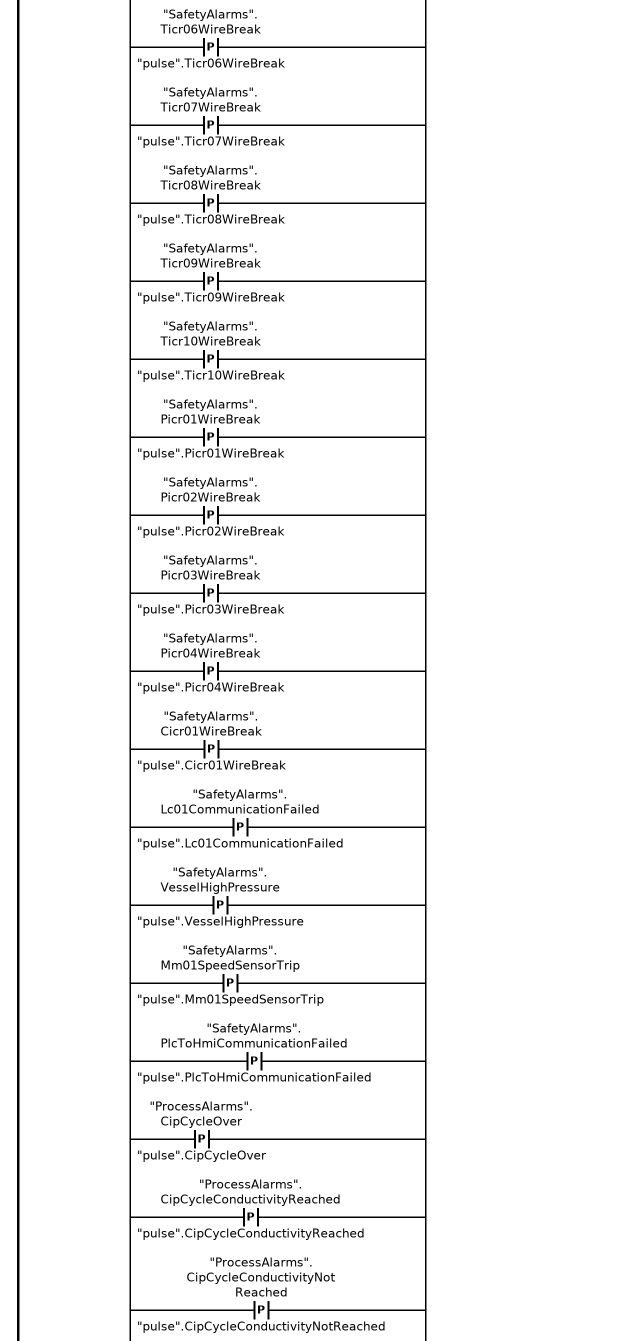
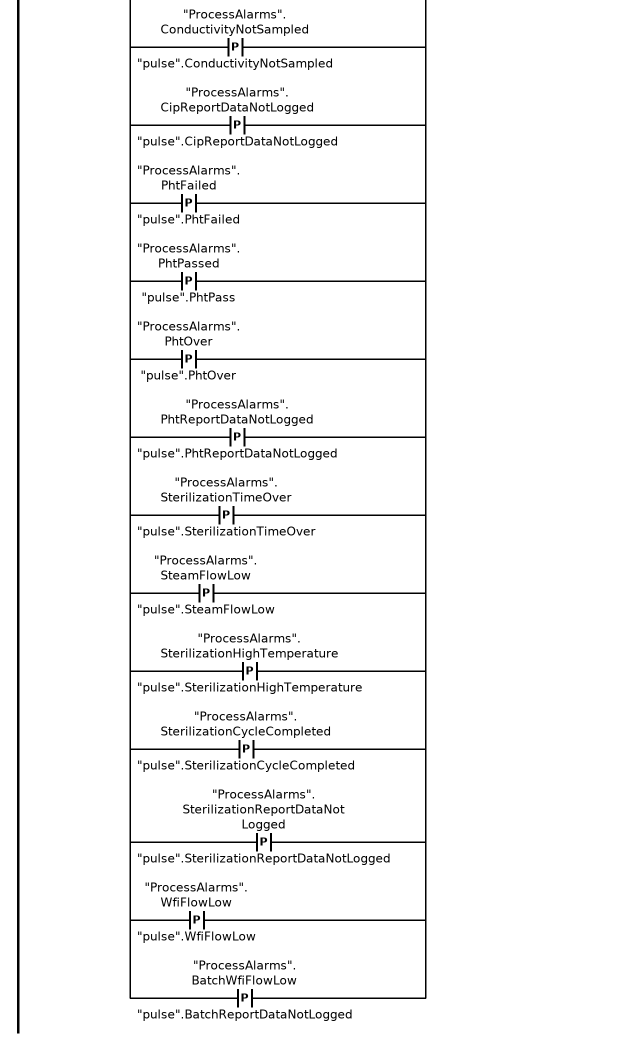
   RUNG wire#powerrail
      Contact( "AlwaysTRUE" )
      wire#w1
      P_Contact(operand := "SafetyAlarms".ControlKeyOff, bit := "pulse".ControlKeyOff)
      wire#w2
      S_Coil( "HmiTags".Hooter )
   END_RUNG
   RUNG wire#w1
      P_Contact(operand := "SafetyAlarms".EmergencyStopPressed, bit := "pulse".EmergencyStopPressed)
   END_RUNG wire#w2
   RUNG wire#w1
      P_Contact(operand := "SafetyAlarms".PowerReset, bit := "pulse".PowerReset)
   END_RUNG wire#w2
   RUNG wire#w1
      P_Contact(operand := "SafetyAlarms".CompresseDairPressurelow, bit := "pulse".CompresseDairPressurelow)
   END_RUNG wire#w2
   RUNG wire#w1
      P_Contact(operand := "SafetyAlarms".PowerFailure, bit := "pulse".PowerFailure)
   END_RUNG wire#w2
   RUNG wire#w1
      P_Contact(operand := "SafetyAlarms".PlcRestarted, bit := "pulse".PlcRestarted)
   END_RUNG wire#w2
   RUNG wire#w1
      P_Contact(operand := "SafetyAlarms".Mm01FeedbackTrip, bit := "pulse".Mm01FeedbackTrip)
   END_RUNG wire#w2
   RUNG wire#w1
      P_Contact(operand := "SafetyAlarms".Cp01FeedbackTrip, bit := "pulse".Cp01FeedbackTrip)
   END_RUNG wire#w2
   RUNG wire#w1
      P_Contact(operand := "SafetyAlarms".Mm01OverloadTrip, bit := "pulse".Mm01OverloadTrip)
   END_RUNG wire#w2
   RUNG wire#w1
      P_Contact(operand := "SafetyAlarms".Cp01OverloadTrip, bit := "pulse".Cp01OverloadTrip)
   END_RUNG wire#w2
   RUNG wire#w1
      P_Contact(operand := "SafetyAlarms".MinimumWeightRequiredToStartmm01, bit := "pulse".MinimumWeightRequiredToStartmm01)
   END_RUNG wire#w2
   RUNG wire#w1
      P_Contact(operand := "SafetyAlarms".Ticr01WireBreak, bit := "pulse".Ticr01WireBreak)
   END_RUNG wire#w2
   RUNG wire#w1
      P_Contact(operand := "SafetyAlarms".Ticr02WireBreak, bit := "pulse".Ticr02WireBreak)
   END_RUNG wire#w2
   RUNG wire#w1
      P_Contact(operand := "SafetyAlarms".Ticr03WireBreak, bit := "pulse".Ticr03WireBreak)
   END_RUNG wire#w2
   RUNG wire#w1
      P_Contact(operand := "SafetyAlarms".Ticr04WireBreak, bit := "pulse".Ticr04WireBreak)
   END_RUNG wire#w2
   RUNG wire#w1
      P_Contact(operand := "SafetyAlarms".Ticr05WireBreak, bit := "pulse".Ticr05WireBreak)
   END_RUNG wire#w2
   RUNG wire#w1
      P_Contact(operand := "SafetyAlarms".Ticr06WireBreak, bit := "pulse".Ticr06WireBreak)
   END_RUNG wire#w2
   RUNG wire#w1
      P_Contact(operand := "SafetyAlarms".Ticr07WireBreak, bit := "pulse".Ticr07WireBreak)
   END_RUNG wire#w2
   RUNG wire#w1
      P_Contact(operand := "SafetyAlarms".Ticr08WireBreak, bit := "pulse".Ticr08WireBreak)
   END_RUNG wire#w2
   RUNG wire#w1
      P_Contact(operand := "SafetyAlarms".Ticr09WireBreak, bit := "pulse".Ticr09WireBreak)
   END_RUNG wire#w2
   RUNG wire#w1
      P_Contact(operand := "SafetyAlarms".Ticr10WireBreak, bit := "pulse".Ticr10WireBreak)
   END_RUNG wire#w2
   RUNG wire#w1
      P_Contact(operand := "SafetyAlarms".Picr01WireBreak, bit := "pulse".Picr01WireBreak)
   END_RUNG wire#w2
   RUNG wire#w1
      P_Contact(operand := "SafetyAlarms".Picr02WireBreak, bit := "pulse".Picr02WireBreak)
   END_RUNG wire#w2
   RUNG wire#w1
      P_Contact(operand := "SafetyAlarms".Picr03WireBreak, bit := "pulse".Picr03WireBreak)
   END_RUNG wire#w2
   RUNG wire#w1
      P_Contact(operand := "SafetyAlarms".Picr04WireBreak, bit := "pulse".Picr04WireBreak)
   END_RUNG wire#w2
   RUNG wire#w1
      P_Contact(operand := "SafetyAlarms".Cicr01WireBreak, bit := "pulse".Cicr01WireBreak)
   END_RUNG wire#w2
   RUNG wire#w1
      P_Contact(operand := "SafetyAlarms".Lc01CommunicationFailed, bit := "pulse".Lc01CommunicationFailed)
   END_RUNG wire#w2
   RUNG wire#w1
      P_Contact(operand := "SafetyAlarms".VesselHighPressure, bit := "pulse".VesselHighPressure)
   END_RUNG wire#w2
   RUNG wire#w1
      P_Contact(operand := "SafetyAlarms".Mm01SpeedSensorTrip, bit := "pulse".Mm01SpeedSensorTrip)
   END_RUNG wire#w2
   RUNG wire#w1
      P_Contact(operand := "SafetyAlarms".PlcToHmiCommunicationFailed, bit := "pulse".PlcToHmiCommunicationFailed)
   END_RUNG wire#w2
   RUNG wire#w1
      P_Contact(operand := "ProcessAlarms".CipCycleOver, bit := "pulse".CipCycleOver)
   END_RUNG wire#w2
   RUNG wire#w1
      P_Contact(operand := "ProcessAlarms".CipCycleConductivityReached, bit := "pulse".CipCycleConductivityReached)
   END_RUNG wire#w2
   RUNG wire#w1
      P_Contact(operand := "ProcessAlarms".CipCycleConductivityNotReached, bit := "pulse".CipCycleConductivityNotReached)
   END_RUNG wire#w2
   RUNG wire#w1
      P_Contact(operand := "ProcessAlarms".ConductivityNotSampled, bit := "pulse".ConductivityNotSampled)
   END_RUNG wire#w2
   RUNG wire#w1
      P_Contact(operand := "ProcessAlarms".CipReportDataNotLogged, bit := "pulse".CipReportDataNotLogged)
   END_RUNG wire#w2
   RUNG wire#w1
      P_Contact(operand := "ProcessAlarms".PhtFailed, bit := "pulse".PhtFailed)
   END_RUNG wire#w2
   RUNG wire#w1
      P_Contact(operand := "ProcessAlarms".PhtPassed, bit := "pulse".PhtPass)
   END_RUNG wire#w2
   RUNG wire#w1
      P_Contact(operand := "ProcessAlarms".PhtOver, bit := "pulse".PhtOver)
   END_RUNG wire#w2
   RUNG wire#w1
      P_Contact(operand := "ProcessAlarms".PhtReportDataNotLogged, bit := "pulse".PhtReportDataNotLogged)
   END_RUNG wire#w2
   RUNG wire#w1
      P_Contact(operand := "ProcessAlarms".SterilizationTimeOver, bit := "pulse".SterilizationTimeOver)
   END_RUNG wire#w2
   RUNG wire#w1
      P_Contact(operand := "ProcessAlarms".SteamFlowLow, bit := "pulse".SteamFlowLow)
   END_RUNG wire#w2
   RUNG wire#w1
      P_Contact(operand := "ProcessAlarms".SterilizationHighTemperature, bit := "pulse".SterilizationHighTemperature)
   END_RUNG wire#w2
   RUNG wire#w1
      P_Contact(operand := "ProcessAlarms".SterilizationCycleCompleted, bit := "pulse".SterilizationCycleCompleted)
   END_RUNG wire#w2
   RUNG wire#w1
      P_Contact(operand := "ProcessAlarms".SterilizationReportDataNotLogged, bit := "pulse".SterilizationReportDataNotLogged)
   END_RUNG wire#w2
   RUNG wire#w1
      P_Contact(operand := "ProcessAlarms".WfiFlowLow, bit := "pulse".WfiFlowLow)
   END_RUNG wire#w2
   RUNG wire#w1
      P_Contact(operand := "ProcessAlarms".BatchWfiFlowLow, bit := "pulse".BatchReportDataNotLogged)
   END_RUNG wire#w2
   // the same network as SCL:
   #_w1 := "AlwaysTRUE" AND "SafetyAlarms".ControlKeyOff AND NOT "pulse".ControlKeyOff;   // rising edge of "SafetyAlarms".ControlKeyOff
   "pulse".ControlKeyOff := "SafetyAlarms".ControlKeyOff;
   #_w2 := "AlwaysTRUE" AND "SafetyAlarms".EmergencyStopPressed AND NOT "pulse".EmergencyStopPressed;   // rising edge of "SafetyAlarms".EmergencyStopPressed
   "pulse".EmergencyStopPressed := "SafetyAlarms".EmergencyStopPressed;
   #_w3 := "AlwaysTRUE" AND "SafetyAlarms".PowerReset AND NOT "pulse".PowerReset;   // rising edge of "SafetyAlarms".PowerReset
   "pulse".PowerReset := "SafetyAlarms".PowerReset;
   #_w4 := "AlwaysTRUE" AND "SafetyAlarms".CompresseDairPressurelow AND NOT "pulse".CompresseDairPressurelow;   // rising edge of "SafetyAlarms".CompresseDairPressurelow
   "pulse".CompresseDairPressurelow := "SafetyAlarms".CompresseDairPressurelow;
   #_w5 := "AlwaysTRUE" AND "SafetyAlarms".PowerFailure AND NOT "pulse".PowerFailure;   // rising edge of "SafetyAlarms".PowerFailure
   "pulse".PowerFailure := "SafetyAlarms".PowerFailure;
   #_w6 := "AlwaysTRUE" AND "SafetyAlarms".PlcRestarted AND NOT "pulse".PlcRestarted;   // rising edge of "SafetyAlarms".PlcRestarted
   "pulse".PlcRestarted := "SafetyAlarms".PlcRestarted;
   #_w7 := "AlwaysTRUE" AND "SafetyAlarms".Mm01FeedbackTrip AND NOT "pulse".Mm01FeedbackTrip;   // rising edge of "SafetyAlarms".Mm01FeedbackTrip
   "pulse".Mm01FeedbackTrip := "SafetyAlarms".Mm01FeedbackTrip;
   #_w8 := "AlwaysTRUE" AND "SafetyAlarms".Cp01FeedbackTrip AND NOT "pulse".Cp01FeedbackTrip;   // rising edge of "SafetyAlarms".Cp01FeedbackTrip
   "pulse".Cp01FeedbackTrip := "SafetyAlarms".Cp01FeedbackTrip;
   #_w9 := "AlwaysTRUE" AND "SafetyAlarms".Mm01OverloadTrip AND NOT "pulse".Mm01OverloadTrip;   // rising edge of "SafetyAlarms".Mm01OverloadTrip
   "pulse".Mm01OverloadTrip := "SafetyAlarms".Mm01OverloadTrip;
   #_w10 := "AlwaysTRUE" AND "SafetyAlarms".Cp01OverloadTrip AND NOT "pulse".Cp01OverloadTrip;   // rising edge of "SafetyAlarms".Cp01OverloadTrip
   "pulse".Cp01OverloadTrip := "SafetyAlarms".Cp01OverloadTrip;
   #_w11 := "AlwaysTRUE" AND "SafetyAlarms".MinimumWeightRequiredToStartmm01 AND NOT "pulse".MinimumWeightRequiredToStartmm01;   // rising edge of "SafetyAlarms".MinimumWeightRequiredToStartmm01
   "pulse".MinimumWeightRequiredToStartmm01 := "SafetyAlarms".MinimumWeightRequiredToStartmm01;
   #_w12 := "AlwaysTRUE" AND "SafetyAlarms".Ticr01WireBreak AND NOT "pulse".Ticr01WireBreak;   // rising edge of "SafetyAlarms".Ticr01WireBreak
   "pulse".Ticr01WireBreak := "SafetyAlarms".Ticr01WireBreak;
   #_w13 := "AlwaysTRUE" AND "SafetyAlarms".Ticr02WireBreak AND NOT "pulse".Ticr02WireBreak;   // rising edge of "SafetyAlarms".Ticr02WireBreak
   "pulse".Ticr02WireBreak := "SafetyAlarms".Ticr02WireBreak;
   #_w14 := "AlwaysTRUE" AND "SafetyAlarms".Ticr03WireBreak AND NOT "pulse".Ticr03WireBreak;   // rising edge of "SafetyAlarms".Ticr03WireBreak
   "pulse".Ticr03WireBreak := "SafetyAlarms".Ticr03WireBreak;
   #_w15 := "AlwaysTRUE" AND "SafetyAlarms".Ticr04WireBreak AND NOT "pulse".Ticr04WireBreak;   // rising edge of "SafetyAlarms".Ticr04WireBreak
   "pulse".Ticr04WireBreak := "SafetyAlarms".Ticr04WireBreak;
   #_w16 := "AlwaysTRUE" AND "SafetyAlarms".Ticr05WireBreak AND NOT "pulse".Ticr05WireBreak;   // rising edge of "SafetyAlarms".Ticr05WireBreak
   "pulse".Ticr05WireBreak := "SafetyAlarms".Ticr05WireBreak;
   #_w17 := "AlwaysTRUE" AND "SafetyAlarms".Ticr06WireBreak AND NOT "pulse".Ticr06WireBreak;   // rising edge of "SafetyAlarms".Ticr06WireBreak
   "pulse".Ticr06WireBreak := "SafetyAlarms".Ticr06WireBreak;
   #_w18 := "AlwaysTRUE" AND "SafetyAlarms".Ticr07WireBreak AND NOT "pulse".Ticr07WireBreak;   // rising edge of "SafetyAlarms".Ticr07WireBreak
   "pulse".Ticr07WireBreak := "SafetyAlarms".Ticr07WireBreak;
   #_w19 := "AlwaysTRUE" AND "SafetyAlarms".Ticr08WireBreak AND NOT "pulse".Ticr08WireBreak;   // rising edge of "SafetyAlarms".Ticr08WireBreak
   "pulse".Ticr08WireBreak := "SafetyAlarms".Ticr08WireBreak;
   #_w20 := "AlwaysTRUE" AND "SafetyAlarms".Ticr09WireBreak AND NOT "pulse".Ticr09WireBreak;   // rising edge of "SafetyAlarms".Ticr09WireBreak
   "pulse".Ticr09WireBreak := "SafetyAlarms".Ticr09WireBreak;
   #_w21 := "AlwaysTRUE" AND "SafetyAlarms".Ticr10WireBreak AND NOT "pulse".Ticr10WireBreak;   // rising edge of "SafetyAlarms".Ticr10WireBreak
   "pulse".Ticr10WireBreak := "SafetyAlarms".Ticr10WireBreak;
   #_w22 := "AlwaysTRUE" AND "SafetyAlarms".Picr01WireBreak AND NOT "pulse".Picr01WireBreak;   // rising edge of "SafetyAlarms".Picr01WireBreak
   "pulse".Picr01WireBreak := "SafetyAlarms".Picr01WireBreak;
   #_w23 := "AlwaysTRUE" AND "SafetyAlarms".Picr02WireBreak AND NOT "pulse".Picr02WireBreak;   // rising edge of "SafetyAlarms".Picr02WireBreak
   "pulse".Picr02WireBreak := "SafetyAlarms".Picr02WireBreak;
   #_w24 := "AlwaysTRUE" AND "SafetyAlarms".Picr03WireBreak AND NOT "pulse".Picr03WireBreak;   // rising edge of "SafetyAlarms".Picr03WireBreak
   "pulse".Picr03WireBreak := "SafetyAlarms".Picr03WireBreak;
   #_w25 := "AlwaysTRUE" AND "SafetyAlarms".Picr04WireBreak AND NOT "pulse".Picr04WireBreak;   // rising edge of "SafetyAlarms".Picr04WireBreak
   "pulse".Picr04WireBreak := "SafetyAlarms".Picr04WireBreak;
   #_w26 := "AlwaysTRUE" AND "SafetyAlarms".Cicr01WireBreak AND NOT "pulse".Cicr01WireBreak;   // rising edge of "SafetyAlarms".Cicr01WireBreak
   "pulse".Cicr01WireBreak := "SafetyAlarms".Cicr01WireBreak;
   #_w27 := "AlwaysTRUE" AND "SafetyAlarms".Lc01CommunicationFailed AND NOT "pulse".Lc01CommunicationFailed;   // rising edge of "SafetyAlarms".Lc01CommunicationFailed
   "pulse".Lc01CommunicationFailed := "SafetyAlarms".Lc01CommunicationFailed;
   #_w28 := "AlwaysTRUE" AND "SafetyAlarms".VesselHighPressure AND NOT "pulse".VesselHighPressure;   // rising edge of "SafetyAlarms".VesselHighPressure
   "pulse".VesselHighPressure := "SafetyAlarms".VesselHighPressure;
   #_w29 := "AlwaysTRUE" AND "SafetyAlarms".Mm01SpeedSensorTrip AND NOT "pulse".Mm01SpeedSensorTrip;   // rising edge of "SafetyAlarms".Mm01SpeedSensorTrip
   "pulse".Mm01SpeedSensorTrip := "SafetyAlarms".Mm01SpeedSensorTrip;
   #_w30 := "AlwaysTRUE" AND "SafetyAlarms".PlcToHmiCommunicationFailed AND NOT "pulse".PlcToHmiCommunicationFailed;   // rising edge of "SafetyAlarms".PlcToHmiCommunicationFailed
   "pulse".PlcToHmiCommunicationFailed := "SafetyAlarms".PlcToHmiCommunicationFailed;
   #_w31 := "AlwaysTRUE" AND "ProcessAlarms".CipCycleOver AND NOT "pulse".CipCycleOver;   // rising edge of "ProcessAlarms".CipCycleOver
   "pulse".CipCycleOver := "ProcessAlarms".CipCycleOver;
   #_w32 := "AlwaysTRUE" AND "ProcessAlarms".CipCycleConductivityReached AND NOT "pulse".CipCycleConductivityReached;   // rising edge of "ProcessAlarms".CipCycleConductivityReached
   "pulse".CipCycleConductivityReached := "ProcessAlarms".CipCycleConductivityReached;
   #_w33 := "AlwaysTRUE" AND "ProcessAlarms".CipCycleConductivityNotReached AND NOT "pulse".CipCycleConductivityNotReached;   // rising edge of "ProcessAlarms".CipCycleConductivityNotReached
   "pulse".CipCycleConductivityNotReached := "ProcessAlarms".CipCycleConductivityNotReached;
   #_w34 := "AlwaysTRUE" AND "ProcessAlarms".ConductivityNotSampled AND NOT "pulse".ConductivityNotSampled;   // rising edge of "ProcessAlarms".ConductivityNotSampled
   "pulse".ConductivityNotSampled := "ProcessAlarms".ConductivityNotSampled;
   #_w35 := "AlwaysTRUE" AND "ProcessAlarms".CipReportDataNotLogged AND NOT "pulse".CipReportDataNotLogged;   // rising edge of "ProcessAlarms".CipReportDataNotLogged
   "pulse".CipReportDataNotLogged := "ProcessAlarms".CipReportDataNotLogged;
   #_w36 := "AlwaysTRUE" AND "ProcessAlarms".PhtFailed AND NOT "pulse".PhtFailed;   // rising edge of "ProcessAlarms".PhtFailed
   "pulse".PhtFailed := "ProcessAlarms".PhtFailed;
   #_w37 := "AlwaysTRUE" AND "ProcessAlarms".PhtPassed AND NOT "pulse".PhtPass;   // rising edge of "ProcessAlarms".PhtPassed
   "pulse".PhtPass := "ProcessAlarms".PhtPassed;
   #_w38 := "AlwaysTRUE" AND "ProcessAlarms".PhtOver AND NOT "pulse".PhtOver;   // rising edge of "ProcessAlarms".PhtOver
   "pulse".PhtOver := "ProcessAlarms".PhtOver;
   #_w39 := "AlwaysTRUE" AND "ProcessAlarms".PhtReportDataNotLogged AND NOT "pulse".PhtReportDataNotLogged;   // rising edge of "ProcessAlarms".PhtReportDataNotLogged
   "pulse".PhtReportDataNotLogged := "ProcessAlarms".PhtReportDataNotLogged;
   #_w40 := "AlwaysTRUE" AND "ProcessAlarms".SterilizationTimeOver AND NOT "pulse".SterilizationTimeOver;   // rising edge of "ProcessAlarms".SterilizationTimeOver
   "pulse".SterilizationTimeOver := "ProcessAlarms".SterilizationTimeOver;
   #_w41 := "AlwaysTRUE" AND "ProcessAlarms".SteamFlowLow AND NOT "pulse".SteamFlowLow;   // rising edge of "ProcessAlarms".SteamFlowLow
   "pulse".SteamFlowLow := "ProcessAlarms".SteamFlowLow;
   #_w42 := "AlwaysTRUE" AND "ProcessAlarms".SterilizationHighTemperature AND NOT "pulse".SterilizationHighTemperature;   // rising edge of "ProcessAlarms".SterilizationHighTemperature
   "pulse".SterilizationHighTemperature := "ProcessAlarms".SterilizationHighTemperature;
   #_w43 := "AlwaysTRUE" AND "ProcessAlarms".SterilizationCycleCompleted AND NOT "pulse".SterilizationCycleCompleted;   // rising edge of "ProcessAlarms".SterilizationCycleCompleted
   "pulse".SterilizationCycleCompleted := "ProcessAlarms".SterilizationCycleCompleted;
   #_w44 := "AlwaysTRUE" AND "ProcessAlarms".SterilizationReportDataNotLogged AND NOT "pulse".SterilizationReportDataNotLogged;   // rising edge of "ProcessAlarms".SterilizationReportDataNotLogged
   "pulse".SterilizationReportDataNotLogged := "ProcessAlarms".SterilizationReportDataNotLogged;
   #_w45 := "AlwaysTRUE" AND "ProcessAlarms".WfiFlowLow AND NOT "pulse".WfiFlowLow;   // rising edge of "ProcessAlarms".WfiFlowLow
   "pulse".WfiFlowLow := "ProcessAlarms".WfiFlowLow;
   #_w46 := "AlwaysTRUE" AND "ProcessAlarms".BatchWfiFlowLow AND NOT "pulse".BatchReportDataNotLogged;   // rising edge of "ProcessAlarms".BatchWfiFlowLow
   "pulse".BatchReportDataNotLogged := "ProcessAlarms".BatchWfiFlowLow;
   IF #_w1 OR #_w2 OR #_w3 OR #_w4 OR #_w5 OR #_w6 OR #_w7 OR #_w8 OR #_w9 OR #_w10 OR #_w11 OR #_w12 OR #_w13 OR #_w14 OR #_w15 OR #_w16 OR #_w17 OR #_w18 OR #_w19 OR #_w20 OR #_w21 OR #_w22 OR #_w23 OR #_w24 OR #_w25 OR #_w26 OR #_w27 OR #_w28 OR #_w29 OR #_w30 OR #_w31 OR #_w32 OR #_w33 OR #_w34 OR #_w35 OR #_w36 OR #_w37 OR #_w38 OR #_w39 OR #_w40 OR #_w41 OR #_w42 OR #_w43 OR #_w44 OR #_w45 OR #_w46 THEN
       "HmiTags".Hooter := TRUE;
   END_IF;
END_REGION

REGION Network 31: "HmiTags".Hooter -- reset
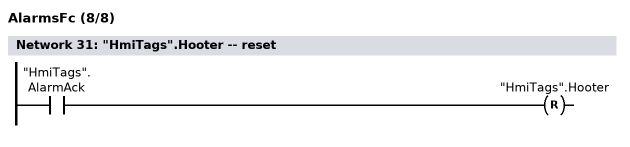
   RUNG wire#powerrail
      Contact( "HmiTags".AlarmAck )
      R_Coil( "HmiTags".Hooter )
   END_RUNG
   // the same network as SCL:
   IF "HmiTags".AlarmAck THEN "HmiTags".Hooter := FALSE; END_IF;
END_REGION
END_FUNCTION
